Staubli VAL3: C2300.pjx

--- C2300.pjx ---
Parameters version=s7.8 stackSize=5000 millimeterUnit=true
Program file=start.pgx
Program file=stop.pgx
Data file=C2300.dtx

--- C2300.dtx ---
public frame fFrmMaster = {x=480, y=190, z=-101.4, rx=2, rz=-90, fatherId=world[0]}
public mdesc mJoint = {accel=50, decel=50, tmax=300, leave=1, reach=1}
mdesc mNomSpeed
public mdesc mNormal = {accel=80, vel=50, decel=50, rmax=9999, tmax=100, leave=2, reach=2}
public num nCompDelta = 0.002
public num nPeak[5]
  [0] = 120
  [1] = 239
  [2] = 303
  [3] = 305
  [4] = 358
public pointRx pDemo[478]
  [0] = {x=50.46, y=-3.411, z=224.779, rx=180, ry=-42.407, rz=-159.872, fatherId=fFrmMaster[0]}
  [1] = {x=4.278, y=-3.411, z=174.216, rx=180, ry=-42.407, rz=-159.872, fatherId=fFrmMaster[0]}
  [2] = {x=4.278, y=-3.411, z=124.216, rx=180, ry=-42.407, rz=-159.872, fatherId=fFrmMaster[0]}
  [3] = {x=3.791, y=1.027, z=124.278, rx=180, ry=-42.212, rz=-156.401, fatherId=fFrmMaster[0]}
  [4] = {x=4.289, y=5.504, z=124.132, rx=180, ry=-42.386, rz=-152.9, fatherId=fFrmMaster[0]}
  [5] = {x=5.782, y=9.947, z=123.764, rx=180, ry=-42.934, rz=-149.41, fatherId=fFrmMaster[0]}
  [6] = {x=8.224, y=14.41, z=123.139, rx=180, ry=-43.84, rz=-145.883, fatherId=fFrmMaster[0]}
  [7] = {x=11.501, y=18.894, z=122.2, rx=180, ry=-45.057, rz=-142.303, fatherId=fFrmMaster[0]}
  [8] = {x=9.824, y=14.861, z=122.959, rx=180, ry=-44.571, rz=-145.522, fatherId=fFrmMaster[0]}
  [9] = {x=8.613, y=10.87, z=123.51, rx=180, ry=-44.23, rz=-148.678, fatherId=fFrmMaster[0]}
  [10] = {x=7.921, y=6.919, z=123.87, rx=180, ry=-44.06, rz=-151.783, fatherId=fFrmMaster[0]}
  [11] = {x=7.772, y=2.954, z=124.054, rx=180, ry=-44.073, rz=-154.884, fatherId=fFrmMaster[0]}
  [12] = {x=8.16, y=-0.997, z=124.064, rx=180, ry=-44.266, rz=-157.97, fatherId=fFrmMaster[0]}
  [13] = {x=7.987, y=2.551, z=124.05, rx=180, ry=-44.179, rz=-155.198, fatherId=fFrmMaster[0]}
  [14] = {x=8.556, y=6.099, z=123.875, rx=180, ry=-44.383, rz=-152.423, fatherId=fFrmMaster[0]}
  [15] = {x=9.86, y=9.613, z=123.529, rx=180, ry=-44.879, rz=-149.664, fatherId=fFrmMaster[0]}
  [16] = {x=11.866, y=13.123, z=122.992, rx=180, ry=-45.653, rz=-146.893, fatherId=fFrmMaster[0]}
  [17] = {x=14.502, y=16.628, z=122.234, rx=180, ry=-46.679, rz=-144.107, fatherId=fFrmMaster[0]}
  [18] = {x=17.496, y=20.822, z=121.12, rx=180, ry=-47.769, rz=-140.737, fatherId=fFrmMaster[0]}
  [19] = {x=20.739, y=24.824, z=119.755, rx=180, ry=-48.936, rz=-137.46, fatherId=fFrmMaster[0]}
  [20] = {x=24.162, y=28.607, z=118.15, rx=180, ry=-50.165, rz=-134.293, fatherId=fFrmMaster[0]}
  [21] = {x=27.716, y=32.196, z=116.305, rx=180, ry=-51.442, rz=-131.213, fatherId=fFrmMaster[0]}
  [22] = {x=31.353, y=35.61, z=114.221, rx=180, ry=-52.756, rz=-128.203, fatherId=fFrmMaster[0]}
  [23] = {x=35.033, y=38.861, z=111.903, rx=180, ry=-54.096, rz=-125.249, fatherId=fFrmMaster[0]}
  [24] = {x=38.719, y=41.93, z=109.366, rx=180, ry=-55.456, rz=-122.365, fatherId=fFrmMaster[0]}
  [25] = {x=42.278, y=44.785, z=106.677, rx=180, ry=-56.784, rz=-119.579, fatherId=fFrmMaster[0]}
  [26] = {x=45.697, y=47.475, z=103.838, rx=180, ry=-58.069, rz=-116.85, fatherId=fFrmMaster[0]}
  [27] = {x=49.013, y=50.027, z=100.834, rx=180, ry=-59.331, rz=-114.154, fatherId=fFrmMaster[0]}
  [28] = {x=44.083, y=48.91, z=103.812, rx=180, ry=-56.777, rz=-115.386, fatherId=fFrmMaster[0]}
  [29] = {x=38.578, y=47.741, z=106.69, rx=180, ry=-54.005, rz=-116.65, fatherId=fFrmMaster[0]}
  [30] = {x=33.15, y=46.43, z=109.226, rx=180, ry=-51.395, rz=-118.029, fatherId=fFrmMaster[0]}
  [31] = {x=27.673, y=45.016, z=111.467, rx=180, ry=-48.846, rz=-119.479, fatherId=fFrmMaster[0]}
  [32] = {x=22.349, y=43.394, z=113.421, rx=180, ry=-46.48, rz=-121.092, fatherId=fFrmMaster[0]}
  [33] = {x=16.731, y=41.59, z=115.171, rx=180, ry=-44.042, rz=-122.836, fatherId=fFrmMaster[0]}
  [34] = {x=10.985, y=39.551, z=116.679, rx=180, ry=-41.623, rz=-124.751, fatherId=fFrmMaster[0]}
  [35] = {x=5.01, y=37.376, z=117.894, rx=180, ry=-39.136, rz=-126.747, fatherId=fFrmMaster[0]}
  [36] = {x=-0.804, y=35.019, z=118.802, rx=180, ry=-36.769, rz=-128.86, fatherId=fFrmMaster[0]}
  [37] = {x=-6.341, y=32.513, z=119.42, rx=180, ry=-34.555, rz=-131.058, fatherId=fFrmMaster[0]}
  [38] = {x=-11.541, y=29.826, z=119.795, rx=180, ry=-32.512, rz=-133.367, fatherId=fFrmMaster[0]}
  [39] = {x=-16.328, y=26.961, z=119.972, rx=180, ry=-30.663, rz=-135.78, fatherId=fFrmMaster[0]}
  [40] = {x=-20.759, y=23.89, z=119.984, rx=180, ry=-28.97, rz=-138.319, fatherId=fFrmMaster[0]}
  [41] = {x=-24.662, y=20.615, z=119.891, rx=180, ry=-27.501, rz=-140.98, fatherId=fFrmMaster[0]}
  [42] = {x=-28.137, y=17.281, z=119.682, rx=180, ry=-26.181, rz=-143.656, fatherId=fFrmMaster[0]}
  [43] = {x=-30.954, y=14.026, z=119.435, rx=180, ry=-25.107, rz=-146.251, fatherId=fFrmMaster[0]}
  [44] = {x=-33.378, y=10.884, z=119.125, rx=180, ry=-24.152, rz=-148.747, fatherId=fFrmMaster[0]}
  [45] = {x=-35.18, y=7.837, z=118.856, rx=180, ry=-23.436, rz=-151.164, fatherId=fFrmMaster[0]}
  [46] = {x=-36.701, y=4.771, z=118.561, rx=180, ry=-22.799, rz=-153.585, fatherId=fFrmMaster[0]}
  [47] = {x=-37.634, y=1.68, z=118.351, rx=180, ry=-22.393, rz=-156.021, fatherId=fFrmMaster[0]}
  [48] = {x=-31.685, y=1.329, z=120.133, rx=180, ry=-25.334, rz=-156.276, fatherId=fFrmMaster[0]}
  [49] = {x=-28.486, y=1.091, z=120.955, rx=180, ry=-26.896, rz=-156.452, fatherId=fFrmMaster[0]}
  [50] = {x=-25.13, y=0.851, z=121.716, rx=180, ry=-28.521, rz=-156.629, fatherId=fFrmMaster[0]}
  [51] = {x=-21.648, y=0.56, z=122.401, rx=180, ry=-30.194, rz=-156.845, fatherId=fFrmMaster[0]}
  [52] = {x=-17.999, y=0.268, z=123.005, rx=180, ry=-31.937, rz=-157.062, fatherId=fFrmMaster[0]}
  [53] = {x=-14.2, y=-0.07, z=123.512, rx=180, ry=-33.74, rz=-157.314, fatherId=fFrmMaster[0]}
  [54] = {x=-10.214, y=-0.41, z=123.912, rx=180, ry=-35.624, rz=-157.568, fatherId=fFrmMaster[0]}
  [55] = {x=-6.064, y=-0.79, z=124.188, rx=180, ry=-37.576, rz=-157.852, fatherId=fFrmMaster[0]}
  [56] = {x=-1.901, y=-1.162, z=124.321, rx=180, ry=-39.531, rz=-158.13, fatherId=fFrmMaster[0]}
  [57] = {x=2.184, y=-1.553, z=124.312, rx=180, ry=-41.448, rz=-158.423, fatherId=fFrmMaster[0]}
  [58] = {x=6.214, y=-1.935, z=124.167, rx=180, ry=-43.341, rz=-158.71, fatherId=fFrmMaster[0]}
  [59] = {x=10.181, y=-2.334, z=123.892, rx=180, ry=-45.206, rz=-159.01, fatherId=fFrmMaster[0]}
  [60] = {x=14.101, y=-2.726, z=123.491, rx=180, ry=-47.055, rz=-159.305, fatherId=fFrmMaster[0]}
  [61] = {x=17.978, y=-3.133, z=122.966, rx=180, ry=-48.89, rz=-159.612, fatherId=fFrmMaster[0]}
  [62] = {x=21.827, y=-3.535, z=122.317, rx=180, ry=-50.72, rz=-159.914, fatherId=fFrmMaster[0]}
  [63] = {x=25.648, y=-3.944, z=121.544, rx=180, ry=-52.547, rz=-160.223, fatherId=fFrmMaster[0]}
  [64] = {x=29.434, y=-4.346, z=120.65, rx=180, ry=-54.37, rz=-160.526, fatherId=fFrmMaster[0]}
  [65] = {x=33.191, y=-4.75, z=119.634, rx=180, ry=-56.193, rz=-160.831, fatherId=fFrmMaster[0]}
  [66] = {x=36.907, y=-5.147, z=118.499, rx=180, ry=-58.013, rz=-161.131, fatherId=fFrmMaster[0]}
  [67] = {x=36.9, y=-1.421, z=118.608, rx=180, ry=-58.063, rz=-158.213, fatherId=fFrmMaster[0]}
  [68] = {x=36.824, y=2.407, z=118.608, rx=180, ry=-58.029, rz=-155.227, fatherId=fFrmMaster[0]}
  [69] = {x=36.718, y=6.276, z=118.48, rx=180, ry=-57.927, rz=-152.208, fatherId=fFrmMaster[0]}
  [70] = {x=36.616, y=10.149, z=118.211, rx=180, ry=-57.771, rz=-149.173, fatherId=fFrmMaster[0]}
  [71] = {x=36.51, y=14.016, z=117.804, rx=180, ry=-57.557, rz=-146.122, fatherId=fFrmMaster[0]}
  [72] = {x=37.169, y=16.535, z=117.228, rx=180, ry=-57.751, rz=-144.116, fatherId=fFrmMaster[0]}
  [73] = {x=38.02, y=19.029, z=116.525, rx=180, ry=-58.02, rz=-142.115, fatherId=fFrmMaster[0]}
  [74] = {x=38.787, y=21.476, z=115.79, rx=180, ry=-58.228, rz=-140.133, fatherId=fFrmMaster[0]}
  [75] = {x=39.708, y=23.854, z=114.947, rx=180, ry=-58.501, rz=-138.184, fatherId=fFrmMaster[0]}
  [76] = {x=40.535, y=26.179, z=114.082, rx=180, ry=-58.709, rz=-136.254, fatherId=fFrmMaster[0]}
  [77] = {x=41.497, y=28.44, z=113.115, rx=180, ry=-58.976, rz=-134.351, fatherId=fFrmMaster[0]}
  [78] = {x=42.362, y=30.659, z=112.13, rx=180, ry=-59.176, rz=-132.457, fatherId=fFrmMaster[0]}
  [79] = {x=43.343, y=32.818, z=111.05, rx=180, ry=-59.428, rz=-130.584, fatherId=fFrmMaster[0]}
  [80] = {x=44.221, y=34.939, z=109.958, rx=180, ry=-59.61, rz=-128.715, fatherId=fFrmMaster[0]}
  [81] = {x=45.196, y=37.004, z=108.778, rx=180, ry=-59.834, rz=-126.861, fatherId=fFrmMaster[0]}
  [82] = {x=46.064, y=39.037, z=107.59, rx=180, ry=-59.985, rz=-125.002, fatherId=fFrmMaster[0]}
  [83] = {x=47.013, y=41.002, z=106.326, rx=180, ry=-60.173, rz=-123.166, fatherId=fFrmMaster[0]}
  [84] = {x=47.863, y=42.921, z=105.062, rx=180, ry=-60.293, rz=-121.334, fatherId=fFrmMaster[0]}
  [85] = {x=48.809, y=44.772, z=103.716, rx=180, ry=-60.46, rz=-119.524, fatherId=fFrmMaster[0]}
  [86] = {x=49.686, y=46.591, z=102.355, rx=180, ry=-60.572, rz=-117.702, fatherId=fFrmMaster[0]}
  [87] = {x=50.7, y=48.352, z=100.888, rx=180, ry=-60.754, rz=-115.891, fatherId=fFrmMaster[0]}
  [88] = {x=51.727, y=50.068, z=99.369, rx=180, ry=-60.931, rz=-114.077, fatherId=fFrmMaster[0]}
  [89] = {x=52.948, y=51.706, z=97.716, rx=180, ry=-61.221, rz=-112.29, fatherId=fFrmMaster[0]}
  [90] = {x=54.179, y=53.292, z=96.009, rx=180, ry=-61.51, rz=-110.505, fatherId=fFrmMaster[0]}
  [91] = {x=55.616, y=54.796, z=94.148, rx=180, ry=-61.931, rz=-108.75, fatherId=fFrmMaster[0]}
  [92] = {x=52.563, y=54.509, z=96.159, rx=180, ry=-60.128, rz=-109.12, fatherId=fFrmMaster[0]}
  [93] = {x=47.423, y=53.901, z=99.331, rx=180, ry=-57.206, rz=-109.889, fatherId=fFrmMaster[0]}
  [94] = {x=44.683, y=53.582, z=100.858, rx=180, ry=-55.691, rz=-110.285, fatherId=fFrmMaster[0]}
  [95] = {x=41.917, y=53.209, z=102.324, rx=180, ry=-54.209, rz=-110.738, fatherId=fFrmMaster[0]}
  [96] = {x=38.974, y=52.828, z=103.762, rx=180, ry=-52.655, rz=-111.197, fatherId=fFrmMaster[0]}
  [97] = {x=36.005, y=52.436, z=105.108, rx=180, ry=-51.115, rz=-111.665, fatherId=fFrmMaster[0]}
  [98] = {x=33.04, y=52.03, z=106.355, rx=180, ry=-49.603, rz=-112.143, fatherId=fFrmMaster[0]}
  [99] = {x=27.328, y=51.09, z=108.557, rx=180, ry=-46.799, rz=-113.223, fatherId=fFrmMaster[0]}
  [100] = {x=21.384, y=50.082, z=110.477, rx=180, ry=-43.956, rz=-114.355, fatherId=fFrmMaster[0]}
  [101] = {x=18.339, y=49.516, z=111.339, rx=180, ry=-42.539, rz=-114.977, fatherId=fFrmMaster[0]}
  [102] = {x=15.169, y=48.922, z=112.135, rx=180, ry=-41.078, rz=-115.621, fatherId=fFrmMaster[0]}
  [103] = {x=11.868, y=48.297, z=112.858, rx=180, ry=-39.57, rz=-116.289, fatherId=fFrmMaster[0]}
  [104] = {x=8.507, y=47.631, z=113.495, rx=180, ry=-38.055, rz=-116.989, fatherId=fFrmMaster[0]}
  [105] = {x=5.171, y=46.89, z=114.053, rx=180, ry=-36.584, rz=-117.755, fatherId=fFrmMaster[0]}
  [106] = {x=1.817, y=46.093, z=114.527, rx=180, ry=-35.126, rz=-118.565, fatherId=fFrmMaster[0]}
  [107] = {x=-1.542, y=45.234, z=114.917, rx=180, ry=-33.688, rz=-119.423, fatherId=fFrmMaster[0]}
  [108] = {x=-4.897, y=44.308, z=115.225, rx=180, ry=-32.273, rz=-120.333, fatherId=fFrmMaster[0]}
  [109] = {x=-11.566, y=42.2, z=115.614, rx=180, ry=-29.532, rz=-122.352, fatherId=fFrmMaster[0]}
  [110] = {x=-17.965, y=39.906, z=115.675, rx=180, ry=-26.955, rz=-124.491, fatherId=fFrmMaster[0]}
  [111] = {x=-24.031, y=37.42, z=115.459, rx=180, ry=-24.556, rz=-126.753, fatherId=fFrmMaster[0]}
  [112] = {x=-29.593, y=34.771, z=115.041, rx=180, ry=-22.399, rz=-129.107, fatherId=fFrmMaster[0]}
  [113] = {x=-34.725, y=31.939, z=114.463, rx=180, ry=-20.436, rz=-131.569, fatherId=fFrmMaster[0]}
  [114] = {x=-39.297, y=28.891, z=113.822, rx=180, ry=-18.731, rz=-134.16, fatherId=fFrmMaster[0]}
  [115] = {x=-43.448, y=25.6, z=113.12, rx=180, ry=-17.202, rz=-136.9, fatherId=fFrmMaster[0]}
  [116] = {x=-47.036, y=22.037, z=112.449, rx=180, ry=-15.915, rz=-139.808, fatherId=fFrmMaster[0]}
  [117] = {x=-50.183, y=18.336, z=111.758, rx=180, ry=-14.774, rz=-142.782, fatherId=fFrmMaster[0]}
  [118] = {x=-52.715, y=14.806, z=111.116, rx=180, ry=-13.835, rz=-145.601, fatherId=fFrmMaster[0]}
  [119] = {x=-52.715, y=14.806, z=161.116, rx=180, ry=-13.835, rz=-145.601, fatherId=fFrmMaster[0]}
  [120] = {x=4.278, y=3.411, z=174.216, rx=180, ry=-42.407, rz=159.872, fatherId=fFrmMaster[0]}
  [121] = {x=4.278, y=3.411, z=124.216, rx=180, ry=-42.407, rz=159.872, fatherId=fFrmMaster[0]}
  [122] = {x=3.791, y=-1.027, z=124.278, rx=180, ry=-42.212, rz=156.401, fatherId=fFrmMaster[0]}
  [123] = {x=4.289, y=-5.504, z=124.132, rx=180, ry=-42.386, rz=152.9, fatherId=fFrmMaster[0]}
  [124] = {x=5.782, y=-9.947, z=123.764, rx=180, ry=-42.934, rz=149.41, fatherId=fFrmMaster[0]}
  [125] = {x=8.224, y=-14.41, z=123.139, rx=180, ry=-43.84, rz=145.883, fatherId=fFrmMaster[0]}
  [126] = {x=11.501, y=-18.894, z=122.2, rx=180, ry=-45.057, rz=142.303, fatherId=fFrmMaster[0]}
  [127] = {x=9.824, y=-14.861, z=122.959, rx=180, ry=-44.571, rz=145.522, fatherId=fFrmMaster[0]}
  [128] = {x=8.613, y=-10.87, z=123.51, rx=180, ry=-44.23, rz=148.678, fatherId=fFrmMaster[0]}
  [129] = {x=7.921, y=-6.919, z=123.87, rx=180, ry=-44.06, rz=151.783, fatherId=fFrmMaster[0]}
  [130] = {x=7.772, y=-2.954, z=124.054, rx=180, ry=-44.073, rz=154.884, fatherId=fFrmMaster[0]}
  [131] = {x=8.16, y=0.997, z=124.064, rx=180, ry=-44.266, rz=157.97, fatherId=fFrmMaster[0]}
  [132] = {x=7.987, y=-2.551, z=124.05, rx=180, ry=-44.179, rz=155.198, fatherId=fFrmMaster[0]}
  [133] = {x=8.556, y=-6.099, z=123.875, rx=180, ry=-44.383, rz=152.423, fatherId=fFrmMaster[0]}
  [134] = {x=9.86, y=-9.613, z=123.529, rx=180, ry=-44.879, rz=149.664, fatherId=fFrmMaster[0]}
  [135] = {x=11.866, y=-13.123, z=122.992, rx=180, ry=-45.653, rz=146.893, fatherId=fFrmMaster[0]}
  [136] = {x=14.502, y=-16.628, z=122.234, rx=180, ry=-46.679, rz=144.107, fatherId=fFrmMaster[0]}
  [137] = {x=17.496, y=-20.822, z=121.12, rx=180, ry=-47.769, rz=140.737, fatherId=fFrmMaster[0]}
  [138] = {x=20.739, y=-24.824, z=119.755, rx=180, ry=-48.936, rz=137.46, fatherId=fFrmMaster[0]}
  [139] = {x=24.162, y=-28.607, z=118.15, rx=180, ry=-50.165, rz=134.293, fatherId=fFrmMaster[0]}
  [140] = {x=27.716, y=-32.196, z=116.305, rx=180, ry=-51.442, rz=131.213, fatherId=fFrmMaster[0]}
  [141] = {x=31.353, y=-35.61, z=114.221, rx=180, ry=-52.756, rz=128.203, fatherId=fFrmMaster[0]}
  [142] = {x=35.033, y=-38.861, z=111.903, rx=180, ry=-54.096, rz=125.249, fatherId=fFrmMaster[0]}
  [143] = {x=38.719, y=-41.93, z=109.366, rx=180, ry=-55.456, rz=122.365, fatherId=fFrmMaster[0]}
  [144] = {x=42.278, y=-44.785, z=106.677, rx=180, ry=-56.784, rz=119.579, fatherId=fFrmMaster[0]}
  [145] = {x=45.697, y=-47.475, z=103.838, rx=180, ry=-58.069, rz=116.85, fatherId=fFrmMaster[0]}
  [146] = {x=49.013, y=-50.027, z=100.834, rx=180, ry=-59.331, rz=114.154, fatherId=fFrmMaster[0]}
  [147] = {x=44.083, y=-48.91, z=103.812, rx=180, ry=-56.777, rz=115.386, fatherId=fFrmMaster[0]}
  [148] = {x=38.578, y=-47.741, z=106.69, rx=180, ry=-54.005, rz=116.65, fatherId=fFrmMaster[0]}
  [149] = {x=33.15, y=-46.43, z=109.226, rx=180, ry=-51.395, rz=118.029, fatherId=fFrmMaster[0]}
  [150] = {x=27.673, y=-45.016, z=111.467, rx=180, ry=-48.846, rz=119.479, fatherId=fFrmMaster[0]}
  [151] = {x=22.349, y=-43.394, z=113.421, rx=180, ry=-46.48, rz=121.092, fatherId=fFrmMaster[0]}
  [152] = {x=16.731, y=-41.59, z=115.171, rx=180, ry=-44.042, rz=122.836, fatherId=fFrmMaster[0]}
  [153] = {x=10.985, y=-39.551, z=116.679, rx=180, ry=-41.623, rz=124.751, fatherId=fFrmMaster[0]}
  [154] = {x=5.01, y=-37.376, z=117.894, rx=180, ry=-39.136, rz=126.747, fatherId=fFrmMaster[0]}
  [155] = {x=-0.804, y=-35.019, z=118.802, rx=180, ry=-36.769, rz=128.86, fatherId=fFrmMaster[0]}
  [156] = {x=-6.341, y=-32.513, z=119.42, rx=180, ry=-34.555, rz=131.058, fatherId=fFrmMaster[0]}
  [157] = {x=-11.541, y=-29.826, z=119.795, rx=180, ry=-32.512, rz=133.367, fatherId=fFrmMaster[0]}
  [158] = {x=-16.328, y=-26.961, z=119.972, rx=180, ry=-30.663, rz=135.78, fatherId=fFrmMaster[0]}
  [159] = {x=-20.759, y=-23.89, z=119.984, rx=180, ry=-28.97, rz=138.319, fatherId=fFrmMaster[0]}
  [160] = {x=-24.662, y=-20.615, z=119.891, rx=180, ry=-27.501, rz=140.98, fatherId=fFrmMaster[0]}
  [161] = {x=-28.137, y=-17.281, z=119.682, rx=180, ry=-26.181, rz=143.656, fatherId=fFrmMaster[0]}
  [162] = {x=-30.954, y=-14.026, z=119.435, rx=180, ry=-25.107, rz=146.251, fatherId=fFrmMaster[0]}
  [163] = {x=-33.378, y=-10.884, z=119.125, rx=180, ry=-24.152, rz=148.747, fatherId=fFrmMaster[0]}
  [164] = {x=-35.18, y=-7.837, z=118.856, rx=180, ry=-23.436, rz=151.164, fatherId=fFrmMaster[0]}
  [165] = {x=-36.701, y=-4.771, z=118.561, rx=180, ry=-22.799, rz=153.585, fatherId=fFrmMaster[0]}
  [166] = {x=-37.634, y=-1.68, z=118.351, rx=180, ry=-22.393, rz=156.021, fatherId=fFrmMaster[0]}
  [167] = {x=-31.685, y=-1.329, z=120.133, rx=180, ry=-25.334, rz=156.276, fatherId=fFrmMaster[0]}
  [168] = {x=-28.486, y=-1.091, z=120.955, rx=180, ry=-26.896, rz=156.452, fatherId=fFrmMaster[0]}
  [169] = {x=-25.13, y=-0.851, z=121.716, rx=180, ry=-28.521, rz=156.629, fatherId=fFrmMaster[0]}
  [170] = {x=-21.648, y=-0.56, z=122.401, rx=180, ry=-30.194, rz=156.845, fatherId=fFrmMaster[0]}
  [171] = {x=-17.999, y=-0.268, z=123.005, rx=180, ry=-31.937, rz=157.062, fatherId=fFrmMaster[0]}
  [172] = {x=-14.2, y=0.07, z=123.512, rx=180, ry=-33.74, rz=157.314, fatherId=fFrmMaster[0]}
  [173] = {x=-10.214, y=0.41, z=123.912, rx=180, ry=-35.624, rz=157.568, fatherId=fFrmMaster[0]}
  [174] = {x=-6.064, y=0.79, z=124.188, rx=180, ry=-37.576, rz=157.852, fatherId=fFrmMaster[0]}
  [175] = {x=-1.901, y=1.162, z=124.321, rx=180, ry=-39.531, rz=158.13, fatherId=fFrmMaster[0]}
  [176] = {x=2.184, y=1.553, z=124.312, rx=180, ry=-41.448, rz=158.423, fatherId=fFrmMaster[0]}
  [177] = {x=6.214, y=1.935, z=124.167, rx=180, ry=-43.341, rz=158.71, fatherId=fFrmMaster[0]}
  [178] = {x=10.181, y=2.334, z=123.892, rx=180, ry=-45.206, rz=159.01, fatherId=fFrmMaster[0]}
  [179] = {x=14.101, y=2.726, z=123.491, rx=180, ry=-47.055, rz=159.305, fatherId=fFrmMaster[0]}
  [180] = {x=17.978, y=3.133, z=122.966, rx=180, ry=-48.89, rz=159.612, fatherId=fFrmMaster[0]}
  [181] = {x=21.827, y=3.535, z=122.317, rx=180, ry=-50.72, rz=159.914, fatherId=fFrmMaster[0]}
  [182] = {x=25.648, y=3.944, z=121.544, rx=180, ry=-52.547, rz=160.223, fatherId=fFrmMaster[0]}
  [183] = {x=29.434, y=4.346, z=120.65, rx=180, ry=-54.37, rz=160.526, fatherId=fFrmMaster[0]}
  [184] = {x=33.191, y=4.75, z=119.634, rx=180, ry=-56.193, rz=160.831, fatherId=fFrmMaster[0]}
  [185] = {x=36.907, y=5.147, z=118.499, rx=180, ry=-58.013, rz=161.131, fatherId=fFrmMaster[0]}
  [186] = {x=36.9, y=1.421, z=118.608, rx=180, ry=-58.063, rz=158.213, fatherId=fFrmMaster[0]}
  [187] = {x=36.824, y=-2.407, z=118.608, rx=180, ry=-58.029, rz=155.227, fatherId=fFrmMaster[0]}
  [188] = {x=36.718, y=-6.276, z=118.48, rx=180, ry=-57.927, rz=152.208, fatherId=fFrmMaster[0]}
  [189] = {x=36.616, y=-10.149, z=118.211, rx=180, ry=-57.771, rz=149.173, fatherId=fFrmMaster[0]}
  [190] = {x=36.51, y=-14.016, z=117.804, rx=180, ry=-57.557, rz=146.122, fatherId=fFrmMaster[0]}
  [191] = {x=37.169, y=-16.535, z=117.228, rx=180, ry=-57.751, rz=144.116, fatherId=fFrmMaster[0]}
  [192] = {x=38.02, y=-19.029, z=116.525, rx=180, ry=-58.02, rz=142.115, fatherId=fFrmMaster[0]}
  [193] = {x=38.787, y=-21.476, z=115.79, rx=180, ry=-58.228, rz=140.133, fatherId=fFrmMaster[0]}
  [194] = {x=39.708, y=-23.854, z=114.947, rx=180, ry=-58.501, rz=138.184, fatherId=fFrmMaster[0]}
  [195] = {x=40.535, y=-26.179, z=114.082, rx=180, ry=-58.709, rz=136.254, fatherId=fFrmMaster[0]}
  [196] = {x=41.497, y=-28.44, z=113.115, rx=180, ry=-58.976, rz=134.351, fatherId=fFrmMaster[0]}
  [197] = {x=42.362, y=-30.659, z=112.13, rx=180, ry=-59.176, rz=132.457, fatherId=fFrmMaster[0]}
  [198] = {x=43.343, y=-32.818, z=111.05, rx=180, ry=-59.428, rz=130.584, fatherId=fFrmMaster[0]}
  [199] = {x=44.221, y=-34.939, z=109.958, rx=180, ry=-59.61, rz=128.715, fatherId=fFrmMaster[0]}
  [200] = {x=45.196, y=-37.004, z=108.778, rx=180, ry=-59.834, rz=126.861, fatherId=fFrmMaster[0]}
  [201] = {x=46.064, y=-39.037, z=107.59, rx=180, ry=-59.985, rz=125.002, fatherId=fFrmMaster[0]}
  [202] = {x=47.013, y=-41.002, z=106.326, rx=180, ry=-60.173, rz=123.166, fatherId=fFrmMaster[0]}
  [203] = {x=47.863, y=-42.921, z=105.062, rx=180, ry=-60.293, rz=121.334, fatherId=fFrmMaster[0]}
  [204] = {x=48.809, y=-44.772, z=103.716, rx=180, ry=-60.46, rz=119.524, fatherId=fFrmMaster[0]}
  [205] = {x=49.686, y=-46.591, z=102.355, rx=180, ry=-60.572, rz=117.702, fatherId=fFrmMaster[0]}
  [206] = {x=50.7, y=-48.352, z=100.888, rx=180, ry=-60.754, rz=115.891, fatherId=fFrmMaster[0]}
  [207] = {x=51.727, y=-50.068, z=99.369, rx=180, ry=-60.931, rz=114.077, fatherId=fFrmMaster[0]}
  [208] = {x=52.948, y=-51.706, z=97.716, rx=180, ry=-61.221, rz=112.29, fatherId=fFrmMaster[0]}
  [209] = {x=54.179, y=-53.292, z=96.009, rx=180, ry=-61.51, rz=110.505, fatherId=fFrmMaster[0]}
  [210] = {x=55.616, y=-54.796, z=94.148, rx=180, ry=-61.931, rz=108.75, fatherId=fFrmMaster[0]}
  [211] = {x=52.563, y=-54.509, z=96.159, rx=180, ry=-60.128, rz=109.12, fatherId=fFrmMaster[0]}
  [212] = {x=47.423, y=-53.901, z=99.331, rx=180, ry=-57.206, rz=109.889, fatherId=fFrmMaster[0]}
  [213] = {x=44.683, y=-53.582, z=100.858, rx=180, ry=-55.691, rz=110.285, fatherId=fFrmMaster[0]}
  [214] = {x=41.917, y=-53.209, z=102.324, rx=180, ry=-54.209, rz=110.738, fatherId=fFrmMaster[0]}
  [215] = {x=38.974, y=-52.828, z=103.762, rx=180, ry=-52.655, rz=111.197, fatherId=fFrmMaster[0]}
  [216] = {x=36.005, y=-52.436, z=105.108, rx=180, ry=-51.115, rz=111.665, fatherId=fFrmMaster[0]}
  [217] = {x=33.04, y=-52.03, z=106.355, rx=180, ry=-49.603, rz=112.143, fatherId=fFrmMaster[0]}
  [218] = {x=27.328, y=-51.09, z=108.557, rx=180, ry=-46.799, rz=113.223, fatherId=fFrmMaster[0]}
  [219] = {x=21.384, y=-50.082, z=110.477, rx=180, ry=-43.956, rz=114.355, fatherId=fFrmMaster[0]}
  [220] = {x=18.339, y=-49.516, z=111.339, rx=180, ry=-42.539, rz=114.977, fatherId=fFrmMaster[0]}
  [221] = {x=15.169, y=-48.922, z=112.135, rx=180, ry=-41.078, rz=115.621, fatherId=fFrmMaster[0]}
  [222] = {x=11.868, y=-48.297, z=112.858, rx=180, ry=-39.57, rz=116.289, fatherId=fFrmMaster[0]}
  [223] = {x=8.507, y=-47.631, z=113.495, rx=180, ry=-38.055, rz=116.989, fatherId=fFrmMaster[0]}
  [224] = {x=5.171, y=-46.89, z=114.053, rx=180, ry=-36.584, rz=117.755, fatherId=fFrmMaster[0]}
  [225] = {x=1.817, y=-46.093, z=114.527, rx=180, ry=-35.126, rz=118.565, fatherId=fFrmMaster[0]}
  [226] = {x=-1.542, y=-45.234, z=114.917, rx=180, ry=-33.688, rz=119.423, fatherId=fFrmMaster[0]}
  [227] = {x=-4.897, y=-44.308, z=115.225, rx=180, ry=-32.273, rz=120.333, fatherId=fFrmMaster[0]}
  [228] = {x=-11.566, y=-42.2, z=115.614, rx=180, ry=-29.532, rz=122.352, fatherId=fFrmMaster[0]}
  [229] = {x=-17.965, y=-39.906, z=115.675, rx=180, ry=-26.955, rz=124.491, fatherId=fFrmMaster[0]}
  [230] = {x=-24.031, y=-37.42, z=115.459, rx=180, ry=-24.556, rz=126.753, fatherId=fFrmMaster[0]}
  [231] = {x=-29.593, y=-34.771, z=115.041, rx=180, ry=-22.399, rz=129.107, fatherId=fFrmMaster[0]}
  [232] = {x=-34.725, y=-31.939, z=114.463, rx=180, ry=-20.436, rz=131.569, fatherId=fFrmMaster[0]}
  [233] = {x=-39.297, y=-28.891, z=113.822, rx=180, ry=-18.731, rz=134.16, fatherId=fFrmMaster[0]}
  [234] = {x=-43.448, y=-25.6, z=113.12, rx=180, ry=-17.202, rz=136.9, fatherId=fFrmMaster[0]}
  [235] = {x=-47.036, y=-22.037, z=112.449, rx=180, ry=-15.915, rz=139.808, fatherId=fFrmMaster[0]}
  [236] = {x=-50.183, y=-18.336, z=111.758, rx=180, ry=-14.774, rz=142.782, fatherId=fFrmMaster[0]}
  [237] = {x=-52.715, y=-14.806, z=111.116, rx=180, ry=-13.835, rz=145.601, fatherId=fFrmMaster[0]}
  [238] = {x=-52.715, y=-14.806, z=161.116, rx=180, ry=-13.835, rz=145.601, fatherId=fFrmMaster[0]}
  [239] = {x=4.278, y=-3.411, z=174.216, rx=180, ry=-42.407, rz=20.128, fatherId=fFrmMaster[0]}
  [240] = {x=4.278, y=-3.411, z=124.216, rx=180, ry=-42.407, rz=20.128, fatherId=fFrmMaster[0]}
  [241] = {x=3.791, y=1.027, z=124.278, rx=180, ry=-42.212, rz=23.599, fatherId=fFrmMaster[0]}
  [242] = {x=4.289, y=5.504, z=124.132, rx=180, ry=-42.386, rz=27.1, fatherId=fFrmMaster[0]}
  [243] = {x=5.782, y=9.947, z=123.764, rx=180, ry=-42.934, rz=30.59, fatherId=fFrmMaster[0]}
  [244] = {x=8.224, y=14.41, z=123.139, rx=180, ry=-43.84, rz=34.117, fatherId=fFrmMaster[0]}
  [245] = {x=11.501, y=18.894, z=122.2, rx=180, ry=-45.057, rz=37.697, fatherId=fFrmMaster[0]}
  [246] = {x=9.824, y=14.861, z=122.959, rx=180, ry=-44.571, rz=34.478, fatherId=fFrmMaster[0]}
  [247] = {x=8.613, y=10.87, z=123.51, rx=180, ry=-44.23, rz=31.322, fatherId=fFrmMaster[0]}
  [248] = {x=7.921, y=6.919, z=123.87, rx=180, ry=-44.06, rz=28.217, fatherId=fFrmMaster[0]}
  [249] = {x=7.772, y=2.954, z=124.054, rx=180, ry=-44.073, rz=25.116, fatherId=fFrmMaster[0]}
  [250] = {x=8.16, y=-0.997, z=124.064, rx=180, ry=-44.266, rz=22.03, fatherId=fFrmMaster[0]}
  [251] = {x=7.987, y=2.551, z=124.05, rx=180, ry=-44.179, rz=24.802, fatherId=fFrmMaster[0]}
  [252] = {x=8.556, y=6.099, z=123.875, rx=180, ry=-44.383, rz=27.577, fatherId=fFrmMaster[0]}
  [253] = {x=9.86, y=9.613, z=123.529, rx=180, ry=-44.879, rz=30.336, fatherId=fFrmMaster[0]}
  [254] = {x=11.866, y=13.123, z=122.992, rx=180, ry=-45.653, rz=33.107, fatherId=fFrmMaster[0]}
  [255] = {x=14.502, y=16.628, z=122.234, rx=180, ry=-46.679, rz=35.893, fatherId=fFrmMaster[0]}
  [256] = {x=17.496, y=20.822, z=121.12, rx=180, ry=-47.769, rz=39.263, fatherId=fFrmMaster[0]}
  [257] = {x=20.739, y=24.824, z=119.755, rx=180, ry=-48.936, rz=42.54, fatherId=fFrmMaster[0]}
  [258] = {x=24.162, y=28.607, z=118.15, rx=180, ry=-50.165, rz=45.707, fatherId=fFrmMaster[0]}
  [259] = {x=27.716, y=32.196, z=116.305, rx=180, ry=-51.442, rz=48.787, fatherId=fFrmMaster[0]}
  [260] = {x=31.353, y=35.61, z=114.221, rx=180, ry=-52.756, rz=51.797, fatherId=fFrmMaster[0]}
  [261] = {x=35.033, y=38.861, z=111.903, rx=180, ry=-54.096, rz=54.751, fatherId=fFrmMaster[0]}
  [262] = {x=38.719, y=41.93, z=109.366, rx=180, ry=-55.456, rz=57.635, fatherId=fFrmMaster[0]}
  [263] = {x=42.278, y=44.785, z=106.677, rx=180, ry=-56.784, rz=60.421, fatherId=fFrmMaster[0]}
  [264] = {x=45.697, y=47.475, z=103.838, rx=180, ry=-58.069, rz=63.15, fatherId=fFrmMaster[0]}
  [265] = {x=49.013, y=50.027, z=100.834, rx=180, ry=-59.331, rz=65.846, fatherId=fFrmMaster[0]}
  [266] = {x=44.083, y=48.91, z=103.812, rx=180, ry=-56.777, rz=64.614, fatherId=fFrmMaster[0]}
  [267] = {x=38.578, y=47.741, z=106.69, rx=180, ry=-54.005, rz=63.35, fatherId=fFrmMaster[0]}
  [268] = {x=33.15, y=46.43, z=109.226, rx=180, ry=-51.395, rz=61.971, fatherId=fFrmMaster[0]}
  [269] = {x=27.673, y=45.016, z=111.467, rx=180, ry=-48.846, rz=60.521, fatherId=fFrmMaster[0]}
  [270] = {x=22.349, y=43.394, z=113.421, rx=180, ry=-46.48, rz=58.908, fatherId=fFrmMaster[0]}
  [271] = {x=16.731, y=41.59, z=115.171, rx=180, ry=-44.042, rz=57.164, fatherId=fFrmMaster[0]}
  [272] = {x=10.985, y=39.551, z=116.679, rx=180, ry=-41.623, rz=55.249, fatherId=fFrmMaster[0]}
  [273] = {x=5.01, y=37.376, z=117.894, rx=180, ry=-39.136, rz=53.253, fatherId=fFrmMaster[0]}
  [274] = {x=-0.804, y=35.019, z=118.802, rx=180, ry=-36.769, rz=51.14, fatherId=fFrmMaster[0]}
  [275] = {x=-6.341, y=32.513, z=119.42, rx=180, ry=-34.555, rz=48.942, fatherId=fFrmMaster[0]}
  [276] = {x=-11.541, y=29.826, z=119.795, rx=180, ry=-32.512, rz=46.633, fatherId=fFrmMaster[0]}
  [277] = {x=-16.328, y=26.961, z=119.972, rx=180, ry=-30.663, rz=44.22, fatherId=fFrmMaster[0]}
  [278] = {x=-20.759, y=23.89, z=119.984, rx=180, ry=-28.97, rz=41.681, fatherId=fFrmMaster[0]}
  [279] = {x=-24.662, y=20.615, z=119.891, rx=180, ry=-27.501, rz=39.02, fatherId=fFrmMaster[0]}
  [280] = {x=-28.137, y=17.281, z=119.682, rx=180, ry=-26.181, rz=36.344, fatherId=fFrmMaster[0]}
  [281] = {x=-30.954, y=14.026, z=119.435, rx=180, ry=-25.107, rz=33.749, fatherId=fFrmMaster[0]}
  [282] = {x=-33.378, y=10.884, z=119.125, rx=180, ry=-24.152, rz=31.253, fatherId=fFrmMaster[0]}
  [283] = {x=-35.18, y=7.837, z=118.856, rx=180, ry=-23.436, rz=28.836, fatherId=fFrmMaster[0]}
  [284] = {x=-36.701, y=4.771, z=118.561, rx=180, ry=-22.799, rz=26.415, fatherId=fFrmMaster[0]}
  [285] = {x=-37.634, y=1.68, z=118.351, rx=180, ry=-22.393, rz=23.979, fatherId=fFrmMaster[0]}
  [286] = {x=-31.685, y=1.329, z=120.133, rx=180, ry=-25.334, rz=23.724, fatherId=fFrmMaster[0]}
  [287] = {x=-28.486, y=1.091, z=120.955, rx=180, ry=-26.896, rz=23.548, fatherId=fFrmMaster[0]}
  [288] = {x=-25.13, y=0.851, z=121.716, rx=180, ry=-28.521, rz=23.371, fatherId=fFrmMaster[0]}
  [289] = {x=-21.648, y=0.56, z=122.401, rx=180, ry=-30.194, rz=23.155, fatherId=fFrmMaster[0]}
  [290] = {x=-17.999, y=0.268, z=123.005, rx=180, ry=-31.937, rz=22.938, fatherId=fFrmMaster[0]}
  [291] = {x=-14.2, y=-0.07, z=123.512, rx=180, ry=-33.74, rz=22.686, fatherId=fFrmMaster[0]}
  [292] = {x=-10.214, y=-0.41, z=123.912, rx=180, ry=-35.624, rz=22.432, fatherId=fFrmMaster[0]}
  [293] = {x=-6.064, y=-0.79, z=124.188, rx=180, ry=-37.576, rz=22.148, fatherId=fFrmMaster[0]}
  [294] = {x=-1.901, y=-1.162, z=124.321, rx=180, ry=-39.531, rz=21.87, fatherId=fFrmMaster[0]}
  [295] = {x=2.184, y=-1.553, z=124.312, rx=180, ry=-41.448, rz=21.577, fatherId=fFrmMaster[0]}
  [296] = {x=6.214, y=-1.935, z=124.167, rx=180, ry=-43.341, rz=21.29, fatherId=fFrmMaster[0]}
  [297] = {x=10.181, y=-2.334, z=123.892, rx=180, ry=-45.206, rz=20.99, fatherId=fFrmMaster[0]}
  [298] = {x=14.101, y=-2.726, z=123.491, rx=180, ry=-47.055, rz=20.695, fatherId=fFrmMaster[0]}
  [299] = {x=17.978, y=-3.133, z=122.966, rx=180, ry=-48.89, rz=20.388, fatherId=fFrmMaster[0]}
  [300] = {x=21.827, y=-3.535, z=122.317, rx=180, ry=-50.72, rz=20.086, fatherId=fFrmMaster[0]}
  [301] = {x=25.648, y=-3.944, z=121.544, rx=180, ry=-52.547, rz=19.777, fatherId=fFrmMaster[0]}
  [302] = {x=29.434, y=-4.346, z=120.65, rx=180, ry=-54.37, rz=19.474, fatherId=fFrmMaster[0]}
  [303] = {x=33.191, y=-4.75, z=119.634, rx=180, ry=-56.193, rz=19.169, fatherId=fFrmMaster[0]}
  [304] = {x=36.907, y=-5.147, z=118.499, rx=180, ry=-58.013, rz=18.869, fatherId=fFrmMaster[0]}
  [305] = {x=36.9, y=-1.421, z=118.608, rx=180, ry=-58.063, rz=21.787, fatherId=fFrmMaster[0]}
  [306] = {x=36.824, y=2.407, z=118.608, rx=180, ry=-58.029, rz=24.773, fatherId=fFrmMaster[0]}
  [307] = {x=36.718, y=6.276, z=118.48, rx=180, ry=-57.927, rz=27.792, fatherId=fFrmMaster[0]}
  [308] = {x=36.616, y=10.149, z=118.211, rx=180, ry=-57.771, rz=30.827, fatherId=fFrmMaster[0]}
  [309] = {x=36.51, y=14.016, z=117.804, rx=180, ry=-57.557, rz=33.878, fatherId=fFrmMaster[0]}
  [310] = {x=37.169, y=16.535, z=117.228, rx=180, ry=-57.751, rz=35.884, fatherId=fFrmMaster[0]}
  [311] = {x=38.02, y=19.029, z=116.525, rx=180, ry=-58.02, rz=37.885, fatherId=fFrmMaster[0]}
  [312] = {x=38.787, y=21.476, z=115.79, rx=180, ry=-58.228, rz=39.867, fatherId=fFrmMaster[0]}
  [313] = {x=39.708, y=23.854, z=114.947, rx=180, ry=-58.501, rz=41.816, fatherId=fFrmMaster[0]}
  [314] = {x=40.535, y=26.179, z=114.082, rx=180, ry=-58.709, rz=43.746, fatherId=fFrmMaster[0]}
  [315] = {x=41.497, y=28.44, z=113.115, rx=180, ry=-58.976, rz=45.649, fatherId=fFrmMaster[0]}
  [316] = {x=42.362, y=30.659, z=112.13, rx=180, ry=-59.176, rz=47.543, fatherId=fFrmMaster[0]}
  [317] = {x=43.343, y=32.818, z=111.05, rx=180, ry=-59.428, rz=49.416, fatherId=fFrmMaster[0]}
  [318] = {x=44.221, y=34.939, z=109.958, rx=180, ry=-59.61, rz=51.285, fatherId=fFrmMaster[0]}
  [319] = {x=45.196, y=37.004, z=108.778, rx=180, ry=-59.834, rz=53.139, fatherId=fFrmMaster[0]}
  [320] = {x=46.064, y=39.037, z=107.59, rx=180, ry=-59.985, rz=54.998, fatherId=fFrmMaster[0]}
  [321] = {x=47.013, y=41.002, z=106.326, rx=180, ry=-60.173, rz=56.834, fatherId=fFrmMaster[0]}
  [322] = {x=47.863, y=42.921, z=105.062, rx=180, ry=-60.293, rz=58.666, fatherId=fFrmMaster[0]}
  [323] = {x=48.809, y=44.772, z=103.716, rx=180, ry=-60.46, rz=60.476, fatherId=fFrmMaster[0]}
  [324] = {x=49.686, y=46.591, z=102.355, rx=180, ry=-60.572, rz=62.298, fatherId=fFrmMaster[0]}
  [325] = {x=50.7, y=48.352, z=100.888, rx=180, ry=-60.754, rz=64.109, fatherId=fFrmMaster[0]}
  [326] = {x=51.727, y=50.068, z=99.369, rx=180, ry=-60.931, rz=65.923, fatherId=fFrmMaster[0]}
  [327] = {x=52.948, y=51.706, z=97.716, rx=180, ry=-61.221, rz=67.71, fatherId=fFrmMaster[0]}
  [328] = {x=54.179, y=53.292, z=96.009, rx=180, ry=-61.51, rz=69.495, fatherId=fFrmMaster[0]}
  [329] = {x=55.616, y=54.796, z=94.148, rx=180, ry=-61.931, rz=71.25, fatherId=fFrmMaster[0]}
  [330] = {x=52.563, y=54.509, z=96.159, rx=180, ry=-60.128, rz=70.88, fatherId=fFrmMaster[0]}
  [331] = {x=47.423, y=53.901, z=99.331, rx=180, ry=-57.206, rz=70.111, fatherId=fFrmMaster[0]}
  [332] = {x=44.683, y=53.582, z=100.858, rx=180, ry=-55.691, rz=69.715, fatherId=fFrmMaster[0]}
  [333] = {x=41.917, y=53.209, z=102.324, rx=180, ry=-54.209, rz=69.262, fatherId=fFrmMaster[0]}
  [334] = {x=38.974, y=52.828, z=103.762, rx=180, ry=-52.655, rz=68.803, fatherId=fFrmMaster[0]}
  [335] = {x=36.005, y=52.436, z=105.108, rx=180, ry=-51.115, rz=68.335, fatherId=fFrmMaster[0]}
  [336] = {x=33.04, y=52.03, z=106.355, rx=180, ry=-49.603, rz=67.857, fatherId=fFrmMaster[0]}
  [337] = {x=27.328, y=51.09, z=108.557, rx=180, ry=-46.799, rz=66.777, fatherId=fFrmMaster[0]}
  [338] = {x=21.384, y=50.082, z=110.477, rx=180, ry=-43.956, rz=65.645, fatherId=fFrmMaster[0]}
  [339] = {x=18.339, y=49.516, z=111.339, rx=180, ry=-42.539, rz=65.023, fatherId=fFrmMaster[0]}
  [340] = {x=15.169, y=48.922, z=112.135, rx=180, ry=-41.078, rz=64.379, fatherId=fFrmMaster[0]}
  [341] = {x=11.868, y=48.297, z=112.858, rx=180, ry=-39.57, rz=63.711, fatherId=fFrmMaster[0]}
  [342] = {x=8.507, y=47.631, z=113.495, rx=180, ry=-38.055, rz=63.011, fatherId=fFrmMaster[0]}
  [343] = {x=5.171, y=46.89, z=114.053, rx=180, ry=-36.584, rz=62.245, fatherId=fFrmMaster[0]}
  [344] = {x=1.817, y=46.093, z=114.527, rx=180, ry=-35.126, rz=61.435, fatherId=fFrmMaster[0]}
  [345] = {x=-1.542, y=45.234, z=114.917, rx=180, ry=-33.688, rz=60.577, fatherId=fFrmMaster[0]}
  [346] = {x=-4.897, y=44.308, z=115.225, rx=180, ry=-32.273, rz=59.667, fatherId=fFrmMaster[0]}
  [347] = {x=-11.566, y=42.2, z=115.614, rx=180, ry=-29.532, rz=57.648, fatherId=fFrmMaster[0]}
  [348] = {x=-17.965, y=39.906, z=115.675, rx=180, ry=-26.955, rz=55.509, fatherId=fFrmMaster[0]}
  [349] = {x=-24.031, y=37.42, z=115.459, rx=180, ry=-24.556, rz=53.247, fatherId=fFrmMaster[0]}
  [350] = {x=-29.593, y=34.771, z=115.041, rx=180, ry=-22.399, rz=50.893, fatherId=fFrmMaster[0]}
  [351] = {x=-34.725, y=31.939, z=114.463, rx=180, ry=-20.436, rz=48.431, fatherId=fFrmMaster[0]}
  [352] = {x=-39.297, y=28.891, z=113.822, rx=180, ry=-18.731, rz=45.84, fatherId=fFrmMaster[0]}
  [353] = {x=-43.448, y=25.6, z=113.12, rx=180, ry=-17.202, rz=43.1, fatherId=fFrmMaster[0]}
  [354] = {x=-47.036, y=22.037, z=112.449, rx=180, ry=-15.915, rz=40.192, fatherId=fFrmMaster[0]}
  [355] = {x=-50.183, y=18.336, z=111.758, rx=180, ry=-14.774, rz=37.218, fatherId=fFrmMaster[0]}
  [356] = {x=-52.715, y=14.806, z=111.116, rx=180, ry=-13.835, rz=34.399, fatherId=fFrmMaster[0]}
  [357] = {x=-52.715, y=14.806, z=161.116, rx=180, ry=-13.835, rz=34.399, fatherId=fFrmMaster[0]}
  [358] = {x=4.278, y=3.411, z=174.216, rx=180, ry=-42.407, rz=-20.128, fatherId=fFrmMaster[0]}
  [359] = {x=4.278, y=3.411, z=124.216, rx=180, ry=-42.407, rz=-20.128, fatherId=fFrmMaster[0]}
  [360] = {x=3.791, y=-1.027, z=124.278, rx=180, ry=-42.212, rz=-23.599, fatherId=fFrmMaster[0]}
  [361] = {x=4.289, y=-5.504, z=124.132, rx=180, ry=-42.386, rz=-27.1, fatherId=fFrmMaster[0]}
  [362] = {x=5.782, y=-9.947, z=123.764, rx=180, ry=-42.934, rz=-30.59, fatherId=fFrmMaster[0]}
  [363] = {x=8.224, y=-14.41, z=123.139, rx=180, ry=-43.84, rz=-34.117, fatherId=fFrmMaster[0]}
  [364] = {x=11.501, y=-18.894, z=122.2, rx=180, ry=-45.057, rz=-37.697, fatherId=fFrmMaster[0]}
  [365] = {x=9.824, y=-14.861, z=122.959, rx=180, ry=-44.571, rz=-34.478, fatherId=fFrmMaster[0]}
  [366] = {x=8.613, y=-10.87, z=123.51, rx=180, ry=-44.23, rz=-31.322, fatherId=fFrmMaster[0]}
  [367] = {x=7.921, y=-6.919, z=123.87, rx=180, ry=-44.06, rz=-28.217, fatherId=fFrmMaster[0]}
  [368] = {x=7.772, y=-2.954, z=124.054, rx=180, ry=-44.073, rz=-25.116, fatherId=fFrmMaster[0]}
  [369] = {x=8.16, y=0.997, z=124.064, rx=180, ry=-44.266, rz=-22.03, fatherId=fFrmMaster[0]}
  [370] = {x=7.987, y=-2.551, z=124.05, rx=180, ry=-44.179, rz=-24.802, fatherId=fFrmMaster[0]}
  [371] = {x=8.556, y=-6.099, z=123.875, rx=180, ry=-44.383, rz=-27.577, fatherId=fFrmMaster[0]}
  [372] = {x=9.86, y=-9.613, z=123.529, rx=180, ry=-44.879, rz=-30.336, fatherId=fFrmMaster[0]}
  [373] = {x=11.866, y=-13.123, z=122.992, rx=180, ry=-45.653, rz=-33.107, fatherId=fFrmMaster[0]}
  [374] = {x=14.502, y=-16.628, z=122.234, rx=180, ry=-46.679, rz=-35.893, fatherId=fFrmMaster[0]}
  [375] = {x=17.496, y=-20.822, z=121.12, rx=180, ry=-47.769, rz=-39.263, fatherId=fFrmMaster[0]}
  [376] = {x=20.739, y=-24.824, z=119.755, rx=180, ry=-48.936, rz=-42.54, fatherId=fFrmMaster[0]}
  [377] = {x=24.162, y=-28.607, z=118.15, rx=180, ry=-50.165, rz=-45.707, fatherId=fFrmMaster[0]}
  [378] = {x=27.716, y=-32.196, z=116.305, rx=180, ry=-51.442, rz=-48.787, fatherId=fFrmMaster[0]}
  [379] = {x=31.353, y=-35.61, z=114.221, rx=180, ry=-52.756, rz=-51.797, fatherId=fFrmMaster[0]}
  [380] = {x=35.033, y=-38.861, z=111.903, rx=180, ry=-54.096, rz=-54.751, fatherId=fFrmMaster[0]}
  [381] = {x=38.719, y=-41.93, z=109.366, rx=180, ry=-55.456, rz=-57.635, fatherId=fFrmMaster[0]}
  [382] = {x=42.278, y=-44.785, z=106.677, rx=180, ry=-56.784, rz=-60.421, fatherId=fFrmMaster[0]}
  [383] = {x=45.697, y=-47.475, z=103.838, rx=180, ry=-58.069, rz=-63.15, fatherId=fFrmMaster[0]}
  [384] = {x=49.013, y=-50.027, z=100.834, rx=180, ry=-59.331, rz=-65.846, fatherId=fFrmMaster[0]}
  [385] = {x=44.083, y=-48.91, z=103.812, rx=180, ry=-56.777, rz=-64.614, fatherId=fFrmMaster[0]}
  [386] = {x=38.578, y=-47.741, z=106.69, rx=180, ry=-54.005, rz=-63.35, fatherId=fFrmMaster[0]}
  [387] = {x=33.15, y=-46.43, z=109.226, rx=180, ry=-51.395, rz=-61.971, fatherId=fFrmMaster[0]}
  [388] = {x=27.673, y=-45.016, z=111.467, rx=180, ry=-48.846, rz=-60.521, fatherId=fFrmMaster[0]}
  [389] = {x=22.349, y=-43.394, z=113.421, rx=180, ry=-46.48, rz=-58.908, fatherId=fFrmMaster[0]}
  [390] = {x=16.731, y=-41.59, z=115.171, rx=180, ry=-44.042, rz=-57.164, fatherId=fFrmMaster[0]}
  [391] = {x=10.985, y=-39.551, z=116.679, rx=180, ry=-41.623, rz=-55.249, fatherId=fFrmMaster[0]}
  [392] = {x=5.01, y=-37.376, z=117.894, rx=180, ry=-39.136, rz=-53.253, fatherId=fFrmMaster[0]}
  [393] = {x=-0.804, y=-35.019, z=118.802, rx=180, ry=-36.769, rz=-51.14, fatherId=fFrmMaster[0]}
  [394] = {x=-6.341, y=-32.513, z=119.42, rx=180, ry=-34.555, rz=-48.942, fatherId=fFrmMaster[0]}
  [395] = {x=-11.541, y=-29.826, z=119.795, rx=180, ry=-32.512, rz=-46.633, fatherId=fFrmMaster[0]}
  [396] = {x=-16.328, y=-26.961, z=119.972, rx=180, ry=-30.663, rz=-44.22, fatherId=fFrmMaster[0]}
  [397] = {x=-20.759, y=-23.89, z=119.984, rx=180, ry=-28.97, rz=-41.681, fatherId=fFrmMaster[0]}
  [398] = {x=-24.662, y=-20.615, z=119.891, rx=180, ry=-27.501, rz=-39.02, fatherId=fFrmMaster[0]}
  [399] = {x=-28.137, y=-17.281, z=119.682, rx=180, ry=-26.181, rz=-36.344, fatherId=fFrmMaster[0]}
  [400] = {x=-30.954, y=-14.026, z=119.435, rx=180, ry=-25.107, rz=-33.749, fatherId=fFrmMaster[0]}
  [401] = {x=-33.378, y=-10.884, z=119.125, rx=180, ry=-24.152, rz=-31.253, fatherId=fFrmMaster[0]}
  [402] = {x=-35.18, y=-7.837, z=118.856, rx=180, ry=-23.436, rz=-28.836, fatherId=fFrmMaster[0]}
  [403] = {x=-36.701, y=-4.771, z=118.561, rx=180, ry=-22.799, rz=-26.415, fatherId=fFrmMaster[0]}
  [404] = {x=-37.634, y=-1.68, z=118.351, rx=180, ry=-22.393, rz=-23.979, fatherId=fFrmMaster[0]}
  [405] = {x=-31.685, y=-1.329, z=120.133, rx=180, ry=-25.334, rz=-23.724, fatherId=fFrmMaster[0]}
  [406] = {x=-28.486, y=-1.091, z=120.955, rx=180, ry=-26.896, rz=-23.548, fatherId=fFrmMaster[0]}
  [407] = {x=-25.13, y=-0.851, z=121.716, rx=180, ry=-28.521, rz=-23.371, fatherId=fFrmMaster[0]}
  [408] = {x=-21.648, y=-0.56, z=122.401, rx=180, ry=-30.194, rz=-23.155, fatherId=fFrmMaster[0]}
  [409] = {x=-17.999, y=-0.268, z=123.005, rx=180, ry=-31.937, rz=-22.938, fatherId=fFrmMaster[0]}
  [410] = {x=-14.2, y=0.07, z=123.512, rx=180, ry=-33.74, rz=-22.686, fatherId=fFrmMaster[0]}
  [411] = {x=-10.214, y=0.41, z=123.912, rx=180, ry=-35.624, rz=-22.432, fatherId=fFrmMaster[0]}
  [412] = {x=-6.064, y=0.79, z=124.188, rx=180, ry=-37.576, rz=-22.148, fatherId=fFrmMaster[0]}
  [413] = {x=-1.901, y=1.162, z=124.321, rx=180, ry=-39.531, rz=-21.87, fatherId=fFrmMaster[0]}
  [414] = {x=2.184, y=1.553, z=124.312, rx=180, ry=-41.448, rz=-21.577, fatherId=fFrmMaster[0]}
  [415] = {x=6.214, y=1.935, z=124.167, rx=180, ry=-43.341, rz=-21.29, fatherId=fFrmMaster[0]}
  [416] = {x=10.181, y=2.334, z=123.892, rx=180, ry=-45.206, rz=-20.99, fatherId=fFrmMaster[0]}
  [417] = {x=14.101, y=2.726, z=123.491, rx=180, ry=-47.055, rz=-20.695, fatherId=fFrmMaster[0]}
  [418] = {x=17.978, y=3.133, z=122.966, rx=180, ry=-48.89, rz=-20.388, fatherId=fFrmMaster[0]}
  [419] = {x=21.827, y=3.535, z=122.317, rx=180, ry=-50.72, rz=-20.086, fatherId=fFrmMaster[0]}
  [420] = {x=25.648, y=3.944, z=121.544, rx=180, ry=-52.547, rz=-19.777, fatherId=fFrmMaster[0]}
  [421] = {x=29.434, y=4.346, z=120.65, rx=180, ry=-54.37, rz=-19.474, fatherId=fFrmMaster[0]}
  [422] = {x=33.191, y=4.75, z=119.634, rx=180, ry=-56.193, rz=-19.169, fatherId=fFrmMaster[0]}
  [423] = {x=36.907, y=5.147, z=118.499, rx=180, ry=-58.013, rz=-18.869, fatherId=fFrmMaster[0]}
  [424] = {x=36.9, y=1.421, z=118.608, rx=180, ry=-58.063, rz=-21.787, fatherId=fFrmMaster[0]}
  [425] = {x=36.824, y=-2.407, z=118.608, rx=180, ry=-58.029, rz=-24.773, fatherId=fFrmMaster[0]}
  [426] = {x=36.718, y=-6.276, z=118.48, rx=180, ry=-57.927, rz=-27.792, fatherId=fFrmMaster[0]}
  [427] = {x=36.616, y=-10.149, z=118.211, rx=180, ry=-57.771, rz=-30.827, fatherId=fFrmMaster[0]}
  [428] = {x=36.51, y=-14.016, z=117.804, rx=180, ry=-57.557, rz=-33.878, fatherId=fFrmMaster[0]}
  [429] = {x=37.169, y=-16.535, z=117.228, rx=180, ry=-57.751, rz=-35.884, fatherId=fFrmMaster[0]}
  [430] = {x=38.02, y=-19.029, z=116.525, rx=180, ry=-58.02, rz=-37.885, fatherId=fFrmMaster[0]}
  [431] = {x=38.787, y=-21.476, z=115.79, rx=180, ry=-58.228, rz=-39.867, fatherId=fFrmMaster[0]}
  [432] = {x=39.708, y=-23.854, z=114.947, rx=180, ry=-58.501, rz=-41.816, fatherId=fFrmMaster[0]}
  [433] = {x=40.535, y=-26.179, z=114.082, rx=180, ry=-58.709, rz=-43.746, fatherId=fFrmMaster[0]}
  [434] = {x=41.497, y=-28.44, z=113.115, rx=180, ry=-58.976, rz=-45.649, fatherId=fFrmMaster[0]}
  [435] = {x=42.362, y=-30.659, z=112.13, rx=180, ry=-59.176, rz=-47.543, fatherId=fFrmMaster[0]}
  [436] = {x=43.343, y=-32.818, z=111.05, rx=180, ry=-59.428, rz=-49.416, fatherId=fFrmMaster[0]}
  [437] = {x=44.221, y=-34.939, z=109.958, rx=180, ry=-59.61, rz=-51.285, fatherId=fFrmMaster[0]}
  [438] = {x=45.196, y=-37.004, z=108.778, rx=180, ry=-59.834, rz=-53.139, fatherId=fFrmMaster[0]}
  [439] = {x=46.064, y=-39.037, z=107.59, rx=180, ry=-59.985, rz=-54.998, fatherId=fFrmMaster[0]}
  [440] = {x=47.013, y=-41.002, z=106.326, rx=180, ry=-60.173, rz=-56.834, fatherId=fFrmMaster[0]}
  [441] = {x=47.863, y=-42.921, z=105.062, rx=180, ry=-60.293, rz=-58.666, fatherId=fFrmMaster[0]}
  [442] = {x=48.809, y=-44.772, z=103.716, rx=180, ry=-60.46, rz=-60.476, fatherId=fFrmMaster[0]}
  [443] = {x=49.686, y=-46.591, z=102.355, rx=180, ry=-60.572, rz=-62.298, fatherId=fFrmMaster[0]}
  [444] = {x=50.7, y=-48.352, z=100.888, rx=180, ry=-60.754, rz=-64.109, fatherId=fFrmMaster[0]}
  [445] = {x=51.727, y=-50.068, z=99.369, rx=180, ry=-60.931, rz=-65.923, fatherId=fFrmMaster[0]}
  [446] = {x=52.948, y=-51.706, z=97.716, rx=180, ry=-61.221, rz=-67.71, fatherId=fFrmMaster[0]}
  [447] = {x=54.179, y=-53.292, z=96.009, rx=180, ry=-61.51, rz=-69.495, fatherId=fFrmMaster[0]}
  [448] = {x=55.616, y=-54.796, z=94.148, rx=180, ry=-61.931, rz=-71.25, fatherId=fFrmMaster[0]}
  [449] = {x=52.563, y=-54.509, z=96.159, rx=180, ry=-60.128, rz=-70.88, fatherId=fFrmMaster[0]}
  [450] = {x=47.423, y=-53.901, z=99.331, rx=180, ry=-57.206, rz=-70.111, fatherId=fFrmMaster[0]}
  [451] = {x=44.683, y=-53.582, z=100.858, rx=180, ry=-55.691, rz=-69.715, fatherId=fFrmMaster[0]}
  [452] = {x=41.917, y=-53.209, z=102.324, rx=180, ry=-54.209, rz=-69.262, fatherId=fFrmMaster[0]}
  [453] = {x=38.974, y=-52.828, z=103.762, rx=180, ry=-52.655, rz=-68.803, fatherId=fFrmMaster[0]}
  [454] = {x=36.005, y=-52.436, z=105.108, rx=180, ry=-51.115, rz=-68.335, fatherId=fFrmMaster[0]}
  [455] = {x=33.04, y=-52.03, z=106.355, rx=180, ry=-49.603, rz=-67.857, fatherId=fFrmMaster[0]}
  [456] = {x=27.328, y=-51.09, z=108.557, rx=180, ry=-46.799, rz=-66.777, fatherId=fFrmMaster[0]}
  [457] = {x=21.384, y=-50.082, z=110.477, rx=180, ry=-43.956, rz=-65.645, fatherId=fFrmMaster[0]}
  [458] = {x=18.339, y=-49.516, z=111.339, rx=180, ry=-42.539, rz=-65.023, fatherId=fFrmMaster[0]}
  [459] = {x=15.169, y=-48.922, z=112.135, rx=180, ry=-41.078, rz=-64.379, fatherId=fFrmMaster[0]}
  [460] = {x=11.868, y=-48.297, z=112.858, rx=180, ry=-39.57, rz=-63.711, fatherId=fFrmMaster[0]}
  [461] = {x=8.507, y=-47.631, z=113.495, rx=180, ry=-38.055, rz=-63.011, fatherId=fFrmMaster[0]}
  [462] = {x=5.171, y=-46.89, z=114.053, rx=180, ry=-36.584, rz=-62.245, fatherId=fFrmMaster[0]}
  [463] = {x=1.817, y=-46.093, z=114.527, rx=180, ry=-35.126, rz=-61.435, fatherId=fFrmMaster[0]}
  [464] = {x=-1.542, y=-45.234, z=114.917, rx=180, ry=-33.688, rz=-60.577, fatherId=fFrmMaster[0]}
  [465] = {x=-4.897, y=-44.308, z=115.225, rx=180, ry=-32.273, rz=-59.667, fatherId=fFrmMaster[0]}
  [466] = {x=-11.566, y=-42.2, z=115.614, rx=180, ry=-29.532, rz=-57.648, fatherId=fFrmMaster[0]}
  [467] = {x=-17.965, y=-39.906, z=115.675, rx=180, ry=-26.955, rz=-55.509, fatherId=fFrmMaster[0]}
  [468] = {x=-24.031, y=-37.42, z=115.459, rx=180, ry=-24.556, rz=-53.247, fatherId=fFrmMaster[0]}
  [469] = {x=-29.593, y=-34.771, z=115.041, rx=180, ry=-22.399, rz=-50.893, fatherId=fFrmMaster[0]}
  [470] = {x=-34.725, y=-31.939, z=114.463, rx=180, ry=-20.436, rz=-48.431, fatherId=fFrmMaster[0]}
  [471] = {x=-39.297, y=-28.891, z=113.822, rx=180, ry=-18.731, rz=-45.84, fatherId=fFrmMaster[0]}
  [472] = {x=-43.448, y=-25.6, z=113.12, rx=180, ry=-17.202, rz=-43.1, fatherId=fFrmMaster[0]}
  [473] = {x=-47.036, y=-22.037, z=112.449, rx=180, ry=-15.915, rz=-40.192, fatherId=fFrmMaster[0]}
  [474] = {x=-50.183, y=-18.336, z=111.758, rx=180, ry=-14.774, rz=-37.218, fatherId=fFrmMaster[0]}
  [475] = {x=-52.715, y=-14.806, z=111.116, rx=180, ry=-13.835, rz=-34.399, fatherId=fFrmMaster[0]}
  [476] = {x=-52.715, y=-14.806, z=161.116, rx=180, ry=-13.835, rz=-34.399, fatherId=fFrmMaster[0]}
  [477] = {x=-39.284, y=-14.806, z=215.651, rx=180, ry=-13.835, rz=-34.399, fatherId=fFrmMaster[0]}
public string sFrameName
public string sJtParameter
public string sPtParameter[478]
  [0] = "-1/-1/-1/-1/-1/-1"
  [1] = "-1/-1/-1/-1/-1/-1"
  [2] = "-1/-1/-1/-1/-1/-1"
  [3] = "-1/-1/-1/-1/-1/-1"
  [4] = "-1/-1/-1/-1/-1/-1"
  [5] = "-1/-1/-1/-1/-1/-1"
  [6] = "-1/-1/-1/-1/-1/-1"
  [7] = "-1/-1/-1/-1/-1/-1"
  [8] = "-1/-1/-1/-1/-1/-1"
  [9] = "-1/-1/-1/-1/-1/-1"
  [10] = "-1/-1/-1/-1/-1/-1"
  [11] = "-1/-1/-1/-1/-1/-1"
  [12] = "-1/-1/-1/-1/-1/-1"
  [13] = "-1/-1/-1/-1/-1/-1"
  [14] = "-1/-1/-1/-1/-1/-1"
  [15] = "-1/-1/-1/-1/-1/-1"
  [16] = "-1/-1/-1/-1/-1/-1"
  [17] = "-1/-1/-1/-1/-1/-1"
  [18] = "-1/-1/-1/-1/-1/-1"
  [19] = "-1/-1/-1/-1/-1/-1"
  [20] = "-1/-1/-1/-1/-1/-1"
  [21] = "-1/-1/-1/-1/-1/-1"
  [22] = "-1/-1/-1/-1/-1/-1"
  [23] = "-1/-1/-1/-1/-1/-1"
  [24] = "-1/-1/-1/-1/-1/-1"
  [25] = "-1/-1/-1/-1/-1/-1"
  [26] = "-1/-1/-1/-1/-1/-1"
  [27] = "-1/-1/-1/-1/-1/-1"
  [28] = "-1/-1/-1/-1/-1/-1"
  [29] = "-1/-1/-1/-1/-1/-1"
  [30] = "-1/-1/-1/-1/-1/-1"
  [31] = "-1/-1/-1/-1/-1/-1"
  [32] = "-1/-1/-1/-1/-1/-1"
  [33] = "-1/-1/-1/-1/-1/-1"
  [34] = "-1/-1/-1/-1/-1/-1"
  [35] = "-1/-1/-1/-1/-1/-1"
  [36] = "-1/-1/-1/-1/-1/-1"
  [37] = "-1/-1/-1/-1/-1/-1"
  [38] = "-1/-1/-1/-1/-1/-1"
  [39] = "-1/-1/-1/-1/-1/-1"
  [40] = "-1/-1/-1/-1/-1/-1"
  [41] = "-1/-1/-1/-1/-1/-1"
  [42] = "-1/-1/-1/-1/-1/-1"
  [43] = "-1/-1/-1/-1/-1/-1"
  [44] = "-1/-1/-1/-1/-1/-1"
  [45] = "-1/-1/-1/-1/-1/-1"
  [46] = "-1/-1/-1/-1/-1/-1"
  [47] = "-1/-1/-1/-1/-1/-1"
  [48] = "-1/-1/-1/-1/-1/-1"
  [49] = "-1/-1/-1/-1/-1/-1"
  [50] = "-1/-1/-1/-1/-1/-1"
  [51] = "-1/-1/-1/-1/-1/-1"
  [52] = "-1/-1/-1/-1/-1/-1"
  [53] = "-1/-1/-1/-1/-1/-1"
  [54] = "-1/-1/-1/-1/-1/-1"
  [55] = "-1/-1/-1/-1/-1/-1"
  [56] = "-1/-1/-1/-1/-1/-1"
  [57] = "-1/-1/-1/-1/-1/-1"
  [58] = "-1/-1/-1/-1/-1/-1"
  [59] = "-1/-1/-1/-1/-1/-1"
  [60] = "-1/-1/-1/-1/-1/-1"
  [61] = "-1/-1/-1/-1/-1/-1"
  [62] = "-1/-1/-1/-1/-1/-1"
  [63] = "-1/-1/-1/-1/-1/-1"
  [64] = "-1/-1/-1/-1/-1/-1"
  [65] = "-1/-1/-1/-1/-1/-1"
  [66] = "-1/-1/-1/-1/-1/-1"
  [67] = "-1/-1/-1/-1/-1/-1"
  [68] = "-1/-1/-1/-1/-1/-1"
  [69] = "-1/-1/-1/-1/-1/-1"
  [70] = "-1/-1/-1/-1/-1/-1"
  [71] = "-1/-1/-1/-1/-1/-1"
  [72] = "-1/-1/-1/-1/-1/-1"
  [73] = "-1/-1/-1/-1/-1/-1"
  [74] = "-1/-1/-1/-1/-1/-1"
  [75] = "-1/-1/-1/-1/-1/-1"
  [76] = "-1/-1/-1/-1/-1/-1"
  [77] = "-1/-1/-1/-1/-1/-1"
  [78] = "-1/-1/-1/-1/-1/-1"
  [79] = "-1/-1/-1/-1/-1/-1"
  [80] = "-1/-1/-1/-1/-1/-1"
  [81] = "-1/-1/-1/-1/-1/-1"
  [82] = "-1/-1/-1/-1/-1/-1"
  [83] = "-1/-1/-1/-1/-1/-1"
  [84] = "-1/-1/-1/-1/-1/-1"
  [85] = "-1/-1/-1/-1/-1/-1"
  [86] = "-1/-1/-1/-1/-1/-1"
  [87] = "-1/-1/-1/-1/-1/-1"
  [88] = "-1/-1/-1/-1/-1/-1"
  [89] = "-1/-1/-1/-1/-1/-1"
  [90] = "-1/-1/-1/-1/-1/-1"
  [91] = "-1/-1/-1/-1/-1/-1"
  [92] = "-1/-1/-1/-1/-1/-1"
  [93] = "-1/-1/-1/-1/-1/-1"
  [94] = "-1/-1/-1/-1/-1/-1"
  [95] = "-1/-1/-1/-1/-1/-1"
  [96] = "-1/-1/-1/-1/-1/-1"
  [97] = "-1/-1/-1/-1/-1/-1"
  [98] = "-1/-1/-1/-1/-1/-1"
  [99] = "-1/-1/-1/-1/-1/-1"
  [100] = "-1/-1/-1/-1/-1/-1"
  [101] = "-1/-1/-1/-1/-1/-1"
  [102] = "-1/-1/-1/-1/-1/-1"
  [103] = "-1/-1/-1/-1/-1/-1"
  [104] = "-1/-1/-1/-1/-1/-1"
  [105] = "-1/-1/-1/-1/-1/-1"
  [106] = "-1/-1/-1/-1/-1/-1"
  [107] = "-1/-1/-1/-1/-1/-1"
  [108] = "-1/-1/-1/-1/-1/-1"
  [109] = "-1/-1/-1/-1/-1/-1"
  [110] = "-1/-1/-1/-1/-1/-1"
  [111] = "-1/-1/-1/-1/-1/-1"
  [112] = "-1/-1/-1/-1/-1/-1"
  [113] = "-1/-1/-1/-1/-1/-1"
  [114] = "-1/-1/-1/-1/-1/-1"
  [115] = "-1/-1/-1/-1/-1/-1"
  [116] = "-1/-1/-1/-1/-1/-1"
  [117] = "-1/-1/-1/-1/-1/-1"
  [118] = "-1/-1/-1/-1/-1/-1"
  [119] = "-1/-1/-1/-1/-1/-1"
  [120] = "-1/-1/-1/-1/-1/-1"
  [121] = "-1/-1/-1/-1/-1/-1"
  [122] = "-1/-1/-1/-1/-1/-1"
  [123] = "-1/-1/-1/-1/-1/-1"
  [124] = "-1/-1/-1/-1/-1/-1"
  [125] = "-1/-1/-1/-1/-1/-1"
  [126] = "-1/-1/-1/-1/-1/-1"
  [127] = "-1/-1/-1/-1/-1/-1"
  [128] = "-1/-1/-1/-1/-1/-1"
  [129] = "-1/-1/-1/-1/-1/-1"
  [130] = "-1/-1/-1/-1/-1/-1"
  [131] = "-1/-1/-1/-1/-1/-1"
  [132] = "-1/-1/-1/-1/-1/-1"
  [133] = "-1/-1/-1/-1/-1/-1"
  [134] = "-1/-1/-1/-1/-1/-1"
  [135] = "-1/-1/-1/-1/-1/-1"
  [136] = "-1/-1/-1/-1/-1/-1"
  [137] = "-1/-1/-1/-1/-1/-1"
  [138] = "-1/-1/-1/-1/-1/-1"
  [139] = "-1/-1/-1/-1/-1/-1"
  [140] = "-1/-1/-1/-1/-1/-1"
  [141] = "-1/-1/-1/-1/-1/-1"
  [142] = "-1/-1/-1/-1/-1/-1"
  [143] = "-1/-1/-1/-1/-1/-1"
  [144] = "-1/-1/-1/-1/-1/-1"
  [145] = "-1/-1/-1/-1/-1/-1"
  [146] = "-1/-1/-1/-1/-1/-1"
  [147] = "-1/-1/-1/-1/-1/-1"
  [148] = "-1/-1/-1/-1/-1/-1"
  [149] = "-1/-1/-1/-1/-1/-1"
  [150] = "-1/-1/-1/-1/-1/-1"
  [151] = "-1/-1/-1/-1/-1/-1"
  [152] = "-1/-1/-1/-1/-1/-1"
  [153] = "-1/-1/-1/-1/-1/-1"
  [154] = "-1/-1/-1/-1/-1/-1"
  [155] = "-1/-1/-1/-1/-1/-1"
  [156] = "-1/-1/-1/-1/-1/-1"
  [157] = "-1/-1/-1/-1/-1/-1"
  [158] = "-1/-1/-1/-1/-1/-1"
  [159] = "-1/-1/-1/-1/-1/-1"
  [160] = "-1/-1/-1/-1/-1/-1"
  [161] = "-1/-1/-1/-1/-1/-1"
  [162] = "-1/-1/-1/-1/-1/-1"
  [163] = "-1/-1/-1/-1/-1/-1"
  [164] = "-1/-1/-1/-1/-1/-1"
  [165] = "-1/-1/-1/-1/-1/-1"
  [166] = "-1/-1/-1/-1/-1/-1"
  [167] = "-1/-1/-1/-1/-1/-1"
  [168] = "-1/-1/-1/-1/-1/-1"
  [169] = "-1/-1/-1/-1/-1/-1"
  [170] = "-1/-1/-1/-1/-1/-1"
  [171] = "-1/-1/-1/-1/-1/-1"
  [172] = "-1/-1/-1/-1/-1/-1"
  [173] = "-1/-1/-1/-1/-1/-1"
  [174] = "-1/-1/-1/-1/-1/-1"
  [175] = "-1/-1/-1/-1/-1/-1"
  [176] = "-1/-1/-1/-1/-1/-1"
  [177] = "-1/-1/-1/-1/-1/-1"
  [178] = "-1/-1/-1/-1/-1/-1"
  [179] = "-1/-1/-1/-1/-1/-1"
  [180] = "-1/-1/-1/-1/-1/-1"
  [181] = "-1/-1/-1/-1/-1/-1"
  [182] = "-1/-1/-1/-1/-1/-1"
  [183] = "-1/-1/-1/-1/-1/-1"
  [184] = "-1/-1/-1/-1/-1/-1"
  [185] = "-1/-1/-1/-1/-1/-1"
  [186] = "-1/-1/-1/-1/-1/-1"
  [187] = "-1/-1/-1/-1/-1/-1"
  [188] = "-1/-1/-1/-1/-1/-1"
  [189] = "-1/-1/-1/-1/-1/-1"
  [190] = "-1/-1/-1/-1/-1/-1"
  [191] = "-1/-1/-1/-1/-1/-1"
  [192] = "-1/-1/-1/-1/-1/-1"
  [193] = "-1/-1/-1/-1/-1/-1"
  [194] = "-1/-1/-1/-1/-1/-1"
  [195] = "-1/-1/-1/-1/-1/-1"
  [196] = "-1/-1/-1/-1/-1/-1"
  [197] = "-1/-1/-1/-1/-1/-1"
  [198] = "-1/-1/-1/-1/-1/-1"
  [199] = "-1/-1/-1/-1/-1/-1"
  [200] = "-1/-1/-1/-1/-1/-1"
  [201] = "-1/-1/-1/-1/-1/-1"
  [202] = "-1/-1/-1/-1/-1/-1"
  [203] = "-1/-1/-1/-1/-1/-1"
  [204] = "-1/-1/-1/-1/-1/-1"
  [205] = "-1/-1/-1/-1/-1/-1"
  [206] = "-1/-1/-1/-1/-1/-1"
  [207] = "-1/-1/-1/-1/-1/-1"
  [208] = "-1/-1/-1/-1/-1/-1"
  [209] = "-1/-1/-1/-1/-1/-1"
  [210] = "-1/-1/-1/-1/-1/-1"
  [211] = "-1/-1/-1/-1/-1/-1"
  [212] = "-1/-1/-1/-1/-1/-1"
  [213] = "-1/-1/-1/-1/-1/-1"
  [214] = "-1/-1/-1/-1/-1/-1"
  [215] = "-1/-1/-1/-1/-1/-1"
  [216] = "-1/-1/-1/-1/-1/-1"
  [217] = "-1/-1/-1/-1/-1/-1"
  [218] = "-1/-1/-1/-1/-1/-1"
  [219] = "-1/-1/-1/-1/-1/-1"
  [220] = "-1/-1/-1/-1/-1/-1"
  [221] = "-1/-1/-1/-1/-1/-1"
  [222] = "-1/-1/-1/-1/-1/-1"
  [223] = "-1/-1/-1/-1/-1/-1"
  [224] = "-1/-1/-1/-1/-1/-1"
  [225] = "-1/-1/-1/-1/-1/-1"
  [226] = "-1/-1/-1/-1/-1/-1"
  [227] = "-1/-1/-1/-1/-1/-1"
  [228] = "-1/-1/-1/-1/-1/-1"
  [229] = "-1/-1/-1/-1/-1/-1"
  [230] = "-1/-1/-1/-1/-1/-1"
  [231] = "-1/-1/-1/-1/-1/-1"
  [232] = "-1/-1/-1/-1/-1/-1"
  [233] = "-1/-1/-1/-1/-1/-1"
  [234] = "-1/-1/-1/-1/-1/-1"
  [235] = "-1/-1/-1/-1/-1/-1"
  [236] = "-1/-1/-1/-1/-1/-1"
  [237] = "-1/-1/-1/-1/-1/-1"
  [238] = "-1/-1/-1/-1/-1/-1"
  [239] = "-1/-1/-1/-1/-1/-1"
  [240] = "-1/-1/-1/-1/-1/-1"
  [241] = "-1/-1/-1/-1/-1/-1"
  [242] = "-1/-1/-1/-1/-1/-1"
  [243] = "-1/-1/-1/-1/-1/-1"
  [244] = "-1/-1/-1/-1/-1/-1"
  [245] = "-1/-1/-1/-1/-1/-1"
  [246] = "-1/-1/-1/-1/-1/-1"
  [247] = "-1/-1/-1/-1/-1/-1"
  [248] = "-1/-1/-1/-1/-1/-1"
  [249] = "-1/-1/-1/-1/-1/-1"
  [250] = "-1/-1/-1/-1/-1/-1"
  [251] = "-1/-1/-1/-1/-1/-1"
  [252] = "-1/-1/-1/-1/-1/-1"
  [253] = "-1/-1/-1/-1/-1/-1"
  [254] = "-1/-1/-1/-1/-1/-1"
  [255] = "-1/-1/-1/-1/-1/-1"
  [256] = "-1/-1/-1/-1/-1/-1"
  [257] = "-1/-1/-1/-1/-1/-1"
  [258] = "-1/-1/-1/-1/-1/-1"
  [259] = "-1/-1/-1/-1/-1/-1"
  [260] = "-1/-1/-1/-1/-1/-1"
  [261] = "-1/-1/-1/-1/-1/-1"
  [262] = "-1/-1/-1/-1/-1/-1"
  [263] = "-1/-1/-1/-1/-1/-1"
  [264] = "-1/-1/-1/-1/-1/-1"
  [265] = "-1/-1/-1/-1/-1/-1"
  [266] = "-1/-1/-1/-1/-1/-1"
  [267] = "-1/-1/-1/-1/-1/-1"
  [268] = "-1/-1/-1/-1/-1/-1"
  [269] = "-1/-1/-1/-1/-1/-1"
  [270] = "-1/-1/-1/-1/-1/-1"
  [271] = "-1/-1/-1/-1/-1/-1"
  [272] = "-1/-1/-1/-1/-1/-1"
  [273] = "-1/-1/-1/-1/-1/-1"
  [274] = "-1/-1/-1/-1/-1/-1"
  [275] = "-1/-1/-1/-1/-1/-1"
  [276] = "-1/-1/-1/-1/-1/-1"
  [277] = "-1/-1/-1/-1/-1/-1"
  [278] = "-1/-1/-1/-1/-1/-1"
  [279] = "-1/-1/-1/-1/-1/-1"
  [280] = "-1/-1/-1/-1/-1/-1"
  [281] = "-1/-1/-1/-1/-1/-1"
  [282] = "-1/-1/-1/-1/-1/-1"
  [283] = "-1/-1/-1/-1/-1/-1"
  [284] = "-1/-1/-1/-1/-1/-1"
  [285] = "-1/-1/-1/-1/-1/-1"
  [286] = "-1/-1/-1/-1/-1/-1"
  [287] = "-1/-1/-1/-1/-1/-1"
  [288] = "-1/-1/-1/-1/-1/-1"
  [289] = "-1/-1/-1/-1/-1/-1"
  [290] = "-1/-1/-1/-1/-1/-1"
  [291] = "-1/-1/-1/-1/-1/-1"
  [292] = "-1/-1/-1/-1/-1/-1"
  [293] = "-1/-1/-1/-1/-1/-1"
  [294] = "-1/-1/-1/-1/-1/-1"
  [295] = "-1/-1/-1/-1/-1/-1"
  [296] = "-1/-1/-1/-1/-1/-1"
  [297] = "-1/-1/-1/-1/-1/-1"
  [298] = "-1/-1/-1/-1/-1/-1"
  [299] = "-1/-1/-1/-1/-1/-1"
  [300] = "-1/-1/-1/-1/-1/-1"
  [301] = "-1/-1/-1/-1/-1/-1"
  [302] = "-1/-1/-1/-1/-1/-1"
  [303] = "-1/-1/-1/-1/-1/-1"
  [304] = "-1/-1/-1/-1/-1/-1"
  [305] = "-1/-1/-1/-1/-1/-1"
  [306] = "-1/-1/-1/-1/-1/-1"
  [307] = "-1/-1/-1/-1/-1/-1"
  [308] = "-1/-1/-1/-1/-1/-1"
  [309] = "-1/-1/-1/-1/-1/-1"
  [310] = "-1/-1/-1/-1/-1/-1"
  [311] = "-1/-1/-1/-1/-1/-1"
  [312] = "-1/-1/-1/-1/-1/-1"
  [313] = "-1/-1/-1/-1/-1/-1"
  [314] = "-1/-1/-1/-1/-1/-1"
  [315] = "-1/-1/-1/-1/-1/-1"
  [316] = "-1/-1/-1/-1/-1/-1"
  [317] = "-1/-1/-1/-1/-1/-1"
  [318] = "-1/-1/-1/-1/-1/-1"
  [319] = "-1/-1/-1/-1/-1/-1"
  [320] = "-1/-1/-1/-1/-1/-1"
  [321] = "-1/-1/-1/-1/-1/-1"
  [322] = "-1/-1/-1/-1/-1/-1"
  [323] = "-1/-1/-1/-1/-1/-1"
  [324] = "-1/-1/-1/-1/-1/-1"
  [325] = "-1/-1/-1/-1/-1/-1"
  [326] = "-1/-1/-1/-1/-1/-1"
  [327] = "-1/-1/-1/-1/-1/-1"
  [328] = "-1/-1/-1/-1/-1/-1"
  [329] = "-1/-1/-1/-1/-1/-1"
  [330] = "-1/-1/-1/-1/-1/-1"
  [331] = "-1/-1/-1/-1/-1/-1"
  [332] = "-1/-1/-1/-1/-1/-1"
  [333] = "-1/-1/-1/-1/-1/-1"
  [334] = "-1/-1/-1/-1/-1/-1"
  [335] = "-1/-1/-1/-1/-1/-1"
  [336] = "-1/-1/-1/-1/-1/-1"
  [337] = "-1/-1/-1/-1/-1/-1"
  [338] = "-1/-1/-1/-1/-1/-1"
  [339] = "-1/-1/-1/-1/-1/-1"
  [340] = "-1/-1/-1/-1/-1/-1"
  [341] = "-1/-1/-1/-1/-1/-1"
  [342] = "-1/-1/-1/-1/-1/-1"
  [343] = "-1/-1/-1/-1/-1/-1"
  [344] = "-1/-1/-1/-1/-1/-1"
  [345] = "-1/-1/-1/-1/-1/-1"
  [346] = "-1/-1/-1/-1/-1/-1"
  [347] = "-1/-1/-1/-1/-1/-1"
  [348] = "-1/-1/-1/-1/-1/-1"
  [349] = "-1/-1/-1/-1/-1/-1"
  [350] = "-1/-1/-1/-1/-1/-1"
  [351] = "-1/-1/-1/-1/-1/-1"
  [352] = "-1/-1/-1/-1/-1/-1"
  [353] = "-1/-1/-1/-1/-1/-1"
  [354] = "-1/-1/-1/-1/-1/-1"
  [355] = "-1/-1/-1/-1/-1/-1"
  [356] = "-1/-1/-1/-1/-1/-1"
  [357] = "-1/-1/-1/-1/-1/-1"
  [358] = "-1/-1/-1/-1/-1/-1"
  [359] = "-1/-1/-1/-1/-1/-1"
  [360] = "-1/-1/-1/-1/-1/-1"
  [361] = "-1/-1/-1/-1/-1/-1"
  [362] = "-1/-1/-1/-1/-1/-1"
  [363] = "-1/-1/-1/-1/-1/-1"
  [364] = "-1/-1/-1/-1/-1/-1"
  [365] = "-1/-1/-1/-1/-1/-1"
  [366] = "-1/-1/-1/-1/-1/-1"
  [367] = "-1/-1/-1/-1/-1/-1"
  [368] = "-1/-1/-1/-1/-1/-1"
  [369] = "-1/-1/-1/-1/-1/-1"
  [370] = "-1/-1/-1/-1/-1/-1"
  [371] = "-1/-1/-1/-1/-1/-1"
  [372] = "-1/-1/-1/-1/-1/-1"
  [373] = "-1/-1/-1/-1/-1/-1"
  [374] = "-1/-1/-1/-1/-1/-1"
  [375] = "-1/-1/-1/-1/-1/-1"
  [376] = "-1/-1/-1/-1/-1/-1"
  [377] = "-1/-1/-1/-1/-1/-1"
  [378] = "-1/-1/-1/-1/-1/-1"
  [379] = "-1/-1/-1/-1/-1/-1"
  [380] = "-1/-1/-1/-1/-1/-1"
  [381] = "-1/-1/-1/-1/-1/-1"
  [382] = "-1/-1/-1/-1/-1/-1"
  [383] = "-1/-1/-1/-1/-1/-1"
  [384] = "-1/-1/-1/-1/-1/-1"
  [385] = "-1/-1/-1/-1/-1/-1"
  [386] = "-1/-1/-1/-1/-1/-1"
  [387] = "-1/-1/-1/-1/-1/-1"
  [388] = "-1/-1/-1/-1/-1/-1"
  [389] = "-1/-1/-1/-1/-1/-1"
  [390] = "-1/-1/-1/-1/-1/-1"
  [391] = "-1/-1/-1/-1/-1/-1"
  [392] = "-1/-1/-1/-1/-1/-1"
  [393] = "-1/-1/-1/-1/-1/-1"
  [394] = "-1/-1/-1/-1/-1/-1"
  [395] = "-1/-1/-1/-1/-1/-1"
  [396] = "-1/-1/-1/-1/-1/-1"
  [397] = "-1/-1/-1/-1/-1/-1"
  [398] = "-1/-1/-1/-1/-1/-1"
  [399] = "-1/-1/-1/-1/-1/-1"
  [400] = "-1/-1/-1/-1/-1/-1"
  [401] = "-1/-1/-1/-1/-1/-1"
  [402] = "-1/-1/-1/-1/-1/-1"
  [403] = "-1/-1/-1/-1/-1/-1"
  [404] = "-1/-1/-1/-1/-1/-1"
  [405] = "-1/-1/-1/-1/-1/-1"
  [406] = "-1/-1/-1/-1/-1/-1"
  [407] = "-1/-1/-1/-1/-1/-1"
  [408] = "-1/-1/-1/-1/-1/-1"
  [409] = "-1/-1/-1/-1/-1/-1"
  [410] = "-1/-1/-1/-1/-1/-1"
  [411] = "-1/-1/-1/-1/-1/-1"
  [412] = "-1/-1/-1/-1/-1/-1"
  [413] = "-1/-1/-1/-1/-1/-1"
  [414] = "-1/-1/-1/-1/-1/-1"
  [415] = "-1/-1/-1/-1/-1/-1"
  [416] = "-1/-1/-1/-1/-1/-1"
  [417] = "-1/-1/-1/-1/-1/-1"
  [418] = "-1/-1/-1/-1/-1/-1"
  [419] = "-1/-1/-1/-1/-1/-1"
  [420] = "-1/-1/-1/-1/-1/-1"
  [421] = "-1/-1/-1/-1/-1/-1"
  [422] = "-1/-1/-1/-1/-1/-1"
  [423] = "-1/-1/-1/-1/-1/-1"
  [424] = "-1/-1/-1/-1/-1/-1"
  [425] = "-1/-1/-1/-1/-1/-1"
  [426] = "-1/-1/-1/-1/-1/-1"
  [427] = "-1/-1/-1/-1/-1/-1"
  [428] = "-1/-1/-1/-1/-1/-1"
  [429] = "-1/-1/-1/-1/-1/-1"
  [430] = "-1/-1/-1/-1/-1/-1"
  [431] = "-1/-1/-1/-1/-1/-1"
  [432] = "-1/-1/-1/-1/-1/-1"
  [433] = "-1/-1/-1/-1/-1/-1"
  [434] = "-1/-1/-1/-1/-1/-1"
  [435] = "-1/-1/-1/-1/-1/-1"
  [436] = "-1/-1/-1/-1/-1/-1"
  [437] = "-1/-1/-1/-1/-1/-1"
  [438] = "-1/-1/-1/-1/-1/-1"
  [439] = "-1/-1/-1/-1/-1/-1"
  [440] = "-1/-1/-1/-1/-1/-1"
  [441] = "-1/-1/-1/-1/-1/-1"
  [442] = "-1/-1/-1/-1/-1/-1"
  [443] = "-1/-1/-1/-1/-1/-1"
  [444] = "-1/-1/-1/-1/-1/-1"
  [445] = "-1/-1/-1/-1/-1/-1"
  [446] = "-1/-1/-1/-1/-1/-1"
  [447] = "-1/-1/-1/-1/-1/-1"
  [448] = "-1/-1/-1/-1/-1/-1"
  [449] = "-1/-1/-1/-1/-1/-1"
  [450] = "-1/-1/-1/-1/-1/-1"
  [451] = "-1/-1/-1/-1/-1/-1"
  [452] = "-1/-1/-1/-1/-1/-1"
  [453] = "-1/-1/-1/-1/-1/-1"
  [454] = "-1/-1/-1/-1/-1/-1"
  [455] = "-1/-1/-1/-1/-1/-1"
  [456] = "-1/-1/-1/-1/-1/-1"
  [457] = "-1/-1/-1/-1/-1/-1"
  [458] = "-1/-1/-1/-1/-1/-1"
  [459] = "-1/-1/-1/-1/-1/-1"
  [460] = "-1/-1/-1/-1/-1/-1"
  [461] = "-1/-1/-1/-1/-1/-1"
  [462] = "-1/-1/-1/-1/-1/-1"
  [463] = "-1/-1/-1/-1/-1/-1"
  [464] = "-1/-1/-1/-1/-1/-1"
  [465] = "-1/-1/-1/-1/-1/-1"
  [466] = "-1/-1/-1/-1/-1/-1"
  [467] = "-1/-1/-1/-1/-1/-1"
  [468] = "-1/-1/-1/-1/-1/-1"
  [469] = "-1/-1/-1/-1/-1/-1"
  [470] = "-1/-1/-1/-1/-1/-1"
  [471] = "-1/-1/-1/-1/-1/-1"
  [472] = "-1/-1/-1/-1/-1/-1"
  [473] = "-1/-1/-1/-1/-1/-1"
  [474] = "-1/-1/-1/-1/-1/-1"
  [475] = "-1/-1/-1/-1/-1/-1"
  [476] = "-1/-1/-1/-1/-1/-1"
  [477] = "-1/-1/-1/-1/-1/-1"
public string sToolName
public tool tTool = {fatherId=flange[0], ioLink=valve1}
